(*

.. <legal notes>

legal notes
=================
| SPDX-FileCopyrightText: © 2026 Oleksandr Tiutyk <trofimich@gmail.com>
| SPDX-License-Identifier: LGPL-3.0-only
| For details check: LGPL-3.0-only_

.. _LGPL-3.0-only: https://www.gnu.org/licenses/lgpl-3.0.en.html

.. </legal notes>

*)

INTERFACE IEvent EXTENDS IObject

{attribute 'monitoring' := 'call'}
PROPERTY Handled : BOOL
GET
END_GET
END_PROPERTY

METHOD SetHandled
END_METHOD

END_INTERFACE

(* stored: Version 1.1.0.1
   Itf IEvent: Id {4290fe22-bbfe-42ca-acfa-29f4b1a003dc}
   Property Handled: Id {887baed9-f1ee-4209-9b76-3b844d59fcde}
   Get Get: Id {4825f4b2-b919-4f9b-9c79-4e4388a5282d}
   Method SetHandled: Id {bf90052d-8d4e-4a65-a834-1f380b97a326} *)
